{attribute addProperty BoxType "EJ7031-0000-0026"}
{attribute addProperty Id "ControlAT %Q*Control_197B7E66162"}
{attribute addProperty CRC "1864676036"}
{attribute addProperty SizeInBites "16"}
{attribute addProperty SizeInBytes "2"}
TYPE STM_Control_6F24B2C4 :
STRUCT
	{attribute addProperty Name "Control"}
	Control AT %Q* : Control_197B7E66;
END_STRUCT
END_TYPE

(* stored: Version 1.2.0.0, ProductVersion 3.1.4024.9
   DUT STM_Control_6F24B2C4: Id {a6fac96d-5e16-4a61-8851-5b1b4515a6c7} *)
